// TIA Portal project "3m-1t-3s" (V16)

(* hardware
DEVICE "S7-1200 station_1"  S7-1200 Station
   slot 0: "Rack_0"  S7-1200 Rack  Rack  V1.0
   slot 1: "PLC_1"  CPU 1212C AC/DC/Rly  6ES7 212-1BE40-0XB0  V4.0
*)

// ===== PLC "PLC_1"  CPU 1212C AC/DC/Rly =====

VAR_GLOBAL   // PLC tag table "Default tag table"
   "start" AT %I0.0 : Bool;
   "stop" AT %I0.1 : Bool;
   "km1" AT %Q0.0 : Bool;
   "km2" AT %Q0.1 : Bool;
   "km3" AT %Q0.2 : Bool;
   "marker loop" AT %M0.0 : Bool;
   "Tag_5" AT %M0.1 : Bool;
   "Tag_6" AT %M0.2 : Bool;
   "Tag_7" AT %M2.0 : Bool;
   "break1" AT %M1.0 : Bool;
   "Tag_1" AT %M0.3 : Bool;
   "Tag_9" AT %M2.1 : Bool;
   "Tag_10" AT %M0.4 : Bool;
   "Tag_11" AT %M0.5 : Bool;
   "km2-run" AT %M1.1 : Bool;
   "Tag_13" AT %M2.2 : Bool;
   "Tag_4" AT %M0.6 : Bool;
   "Break2" AT %M1.2 : Bool;
   "Tag_2" AT %M0.7 : Bool;
   "Tag_8" AT %M1.7 : Bool;
   "Tag_12" AT %M1.6 : Bool;
   "km3-run" AT %M1.3 : Bool;
   "Tag_15" AT %M1.5 : Bool;
   "Tag_14" AT %M2.5 : Bool;
   "Tag_16" AT %M2.6 : Bool;
   "Tag_17" AT %M2.7 : Bool;
   "Break3" AT %M1.4 : Bool;
   "Tag_3" AT %M3.0 : Bool;
   "Tag_18" AT %M3.1 : Bool;
   "Tag_19" AT %M2.3 : Bool;
END_VAR

// folder: System blocks/Program resources

DATA_BLOCK "T1"   // DB1
{ S7_Optimized_Access := 'TRUE' }
AUTHOR : Simatic
FAMILY : IEC
NAME : IEC_TMR
VERSION : 1.0
// stored: InstanceOfName IEC_TIMER
"IEC_TIMER"
BEGIN
END_DATA_BLOCK

// folder: (top level)

ORGANIZATION_BLOCK "Main"   // OB1, LAD, ProgramCycle
TITLE = "Main Program Sweep (Cycle)"
{ S7_Optimized_Access := 'TRUE' }
VERSION : 0.1
   VAR_INPUT
      Initial_Call : Bool;   // Initial call of this OB
      Remanence : Bool;   // =True, if remanent data are available
   END_VAR
   VAR_TEMP   // added for the SCL form of the ladder/FBD networks
      _w1 : Bool;
   END_VAR
BEGIN

REGION Network 1
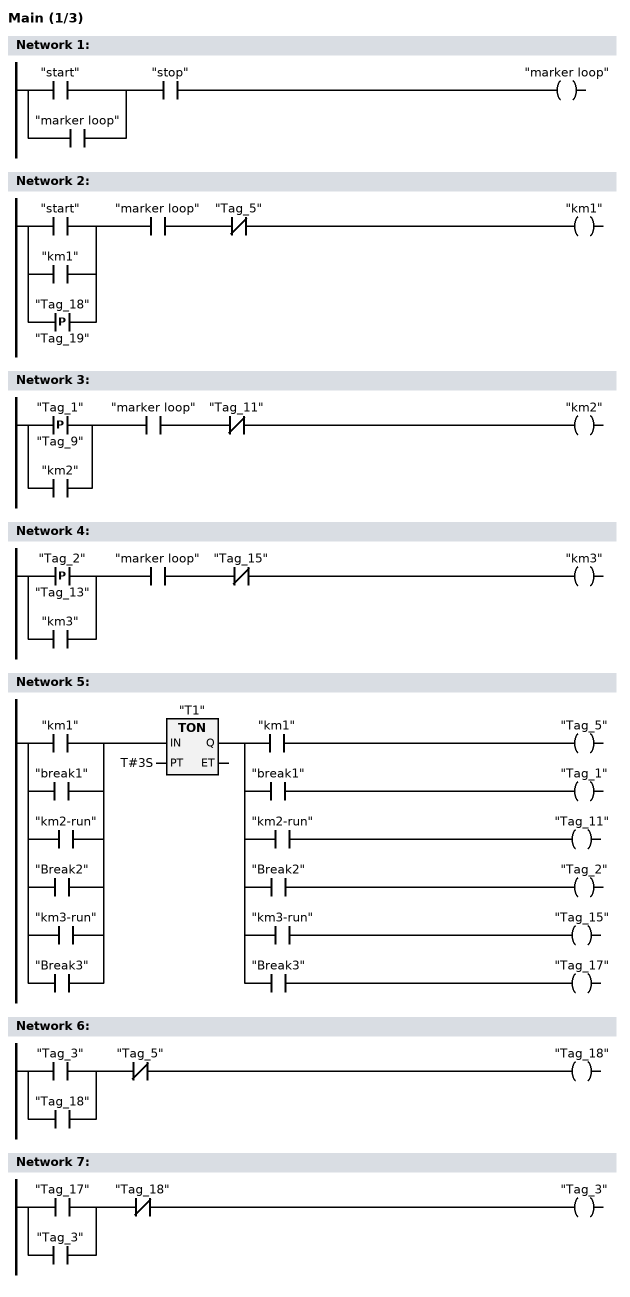
   RUNG wire#powerrail
      Contact( "start" )
      wire#w1
      Contact( "stop" )
      Coil( "marker loop" )
   END_RUNG
   RUNG wire#powerrail
      Contact( "marker loop" )
   END_RUNG wire#w1
   // the same network as SCL:
   "marker loop" := ("start" OR "marker loop") AND "stop";
END_REGION

REGION Network 2
   RUNG wire#powerrail
      Contact( "start" )
      wire#w1
      Contact( "marker loop" )
      I_Contact( "Tag_5" )
      Coil( "km1" )
   END_RUNG
   RUNG wire#powerrail
      Contact( "km1" )
   END_RUNG wire#w1
   RUNG wire#powerrail
      P_Contact(operand := "Tag_18", bit := "Tag_19")
   END_RUNG wire#w1
   // the same network as SCL:
   #_w1 := "Tag_18" AND NOT "Tag_19";   // rising edge of "Tag_18"
   "Tag_19" := "Tag_18";
   "km1" := ("start" OR "km1" OR #_w1) AND "marker loop" AND NOT "Tag_5";
END_REGION

REGION Network 3
   RUNG wire#powerrail
      P_Contact(operand := "Tag_1", bit := "Tag_9")
      wire#w1
      Contact( "marker loop" )
      I_Contact( "Tag_11" )
      Coil( "km2" )
   END_RUNG
   RUNG wire#powerrail
      Contact( "km2" )
   END_RUNG wire#w1
   // the same network as SCL:
   #_w1 := "Tag_1" AND NOT "Tag_9";   // rising edge of "Tag_1"
   "Tag_9" := "Tag_1";
   "km2" := (#_w1 OR "km2") AND "marker loop" AND NOT "Tag_11";
END_REGION

REGION Network 4
   RUNG wire#powerrail
      P_Contact(operand := "Tag_2", bit := "Tag_13")
      wire#w1
      Contact( "marker loop" )
      I_Contact( "Tag_15" )
      Coil( "km3" )
   END_RUNG
   RUNG wire#powerrail
      Contact( "km3" )
   END_RUNG wire#w1
   // the same network as SCL:
   #_w1 := "Tag_2" AND NOT "Tag_13";   // rising edge of "Tag_2"
   "Tag_13" := "Tag_2";
   "km3" := (#_w1 OR "km3") AND "marker loop" AND NOT "Tag_15";
END_REGION

REGION Network 5
   "T1".TON(IN := "km1" OR "break1" OR "km2-run" OR "Break2" OR "km3-run" OR "Break3", PT := T#3S);
   "Tag_5" := "T1".Q AND "km1";
   "Tag_1" := "T1".Q AND "break1";
   "Tag_11" := "T1".Q AND "km2-run";
   "Tag_2" := "T1".Q AND "Break2";
   "Tag_15" := "T1".Q AND "km3-run";
   "Tag_17" := "T1".Q AND "Break3";
END_REGION

REGION Network 6
   RUNG wire#powerrail
      Contact( "Tag_3" )
      wire#w1
      I_Contact( "Tag_5" )
      Coil( "Tag_18" )
   END_RUNG
   RUNG wire#powerrail
      Contact( "Tag_18" )
   END_RUNG wire#w1
   // the same network as SCL:
   "Tag_18" := ("Tag_3" OR "Tag_18") AND NOT "Tag_5";
END_REGION

REGION Network 7
   RUNG wire#powerrail
      Contact( "Tag_17" )
      wire#w1
      I_Contact( "Tag_18" )
      Coil( "Tag_3" )
   END_RUNG
   RUNG wire#powerrail
      Contact( "Tag_3" )
   END_RUNG wire#w1
   // the same network as SCL:
   "Tag_3" := ("Tag_17" OR "Tag_3") AND NOT "Tag_18";
END_REGION

REGION Network 8
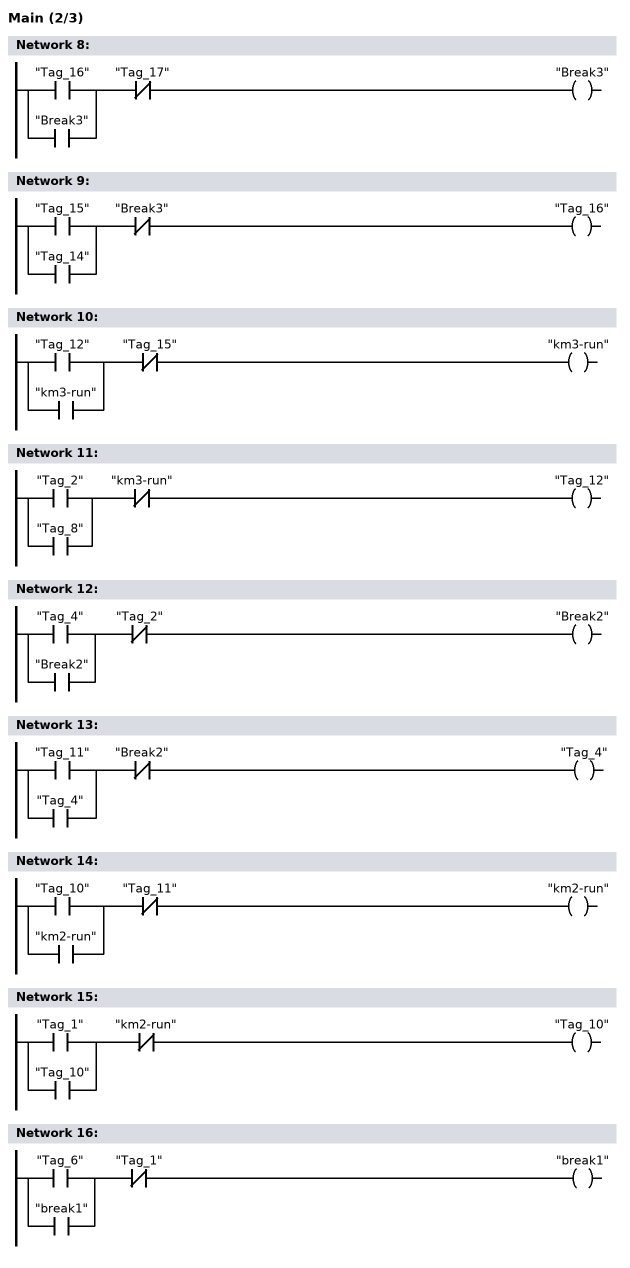
   RUNG wire#powerrail
      Contact( "Tag_16" )
      wire#w1
      I_Contact( "Tag_17" )
      Coil( "Break3" )
   END_RUNG
   RUNG wire#powerrail
      Contact( "Break3" )
   END_RUNG wire#w1
   // the same network as SCL:
   "Break3" := ("Tag_16" OR "Break3") AND NOT "Tag_17";
END_REGION

REGION Network 9
   RUNG wire#powerrail
      Contact( "Tag_15" )
      wire#w1
      I_Contact( "Break3" )
      Coil( "Tag_16" )
   END_RUNG
   RUNG wire#powerrail
      Contact( "Tag_14" )
   END_RUNG wire#w1
   // the same network as SCL:
   "Tag_16" := ("Tag_15" OR "Tag_14") AND NOT "Break3";
END_REGION

REGION Network 10
   RUNG wire#powerrail
      Contact( "Tag_12" )
      wire#w1
      I_Contact( "Tag_15" )
      Coil( "km3-run" )
   END_RUNG
   RUNG wire#powerrail
      Contact( "km3-run" )
   END_RUNG wire#w1
   // the same network as SCL:
   "km3-run" := ("Tag_12" OR "km3-run") AND NOT "Tag_15";
END_REGION

REGION Network 11
   RUNG wire#powerrail
      Contact( "Tag_2" )
      wire#w1
      I_Contact( "km3-run" )
      Coil( "Tag_12" )
   END_RUNG
   RUNG wire#powerrail
      Contact( "Tag_8" )
   END_RUNG wire#w1
   // the same network as SCL:
   "Tag_12" := ("Tag_2" OR "Tag_8") AND NOT "km3-run";
END_REGION

REGION Network 12
   RUNG wire#powerrail
      Contact( "Tag_4" )
      wire#w1
      I_Contact( "Tag_2" )
      Coil( "Break2" )
   END_RUNG
   RUNG wire#powerrail
      Contact( "Break2" )
   END_RUNG wire#w1
   // the same network as SCL:
   "Break2" := ("Tag_4" OR "Break2") AND NOT "Tag_2";
END_REGION

REGION Network 13
   RUNG wire#powerrail
      Contact( "Tag_11" )
      wire#w1
      I_Contact( "Break2" )
      Coil( "Tag_4" )
   END_RUNG
   RUNG wire#powerrail
      Contact( "Tag_4" )
   END_RUNG wire#w1
   // the same network as SCL:
   "Tag_4" := ("Tag_11" OR "Tag_4") AND NOT "Break2";
END_REGION

REGION Network 14
   RUNG wire#powerrail
      Contact( "Tag_10" )
      wire#w1
      I_Contact( "Tag_11" )
      Coil( "km2-run" )
   END_RUNG
   RUNG wire#powerrail
      Contact( "km2-run" )
   END_RUNG wire#w1
   // the same network as SCL:
   "km2-run" := ("Tag_10" OR "km2-run") AND NOT "Tag_11";
END_REGION

REGION Network 15
   RUNG wire#powerrail
      Contact( "Tag_1" )
      wire#w1
      I_Contact( "km2-run" )
      Coil( "Tag_10" )
   END_RUNG
   RUNG wire#powerrail
      Contact( "Tag_10" )
   END_RUNG wire#w1
   // the same network as SCL:
   "Tag_10" := ("Tag_1" OR "Tag_10") AND NOT "km2-run";
END_REGION

REGION Network 16
   RUNG wire#powerrail
      Contact( "Tag_6" )
      wire#w1
      I_Contact( "Tag_1" )
      Coil( "break1" )
   END_RUNG
   RUNG wire#powerrail
      Contact( "break1" )
   END_RUNG wire#w1
   // the same network as SCL:
   "break1" := ("Tag_6" OR "break1") AND NOT "Tag_1";
END_REGION

REGION Network 17
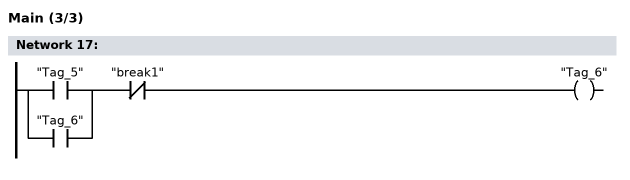
   RUNG wire#powerrail
      Contact( "Tag_5" )
      wire#w1
      I_Contact( "break1" )
      Coil( "Tag_6" )
   END_RUNG
   RUNG wire#powerrail
      Contact( "Tag_6" )
   END_RUNG wire#w1
   // the same network as SCL:
   "Tag_6" := ("Tag_5" OR "Tag_6") AND NOT "break1";
END_REGION
END_ORGANIZATION_BLOCK